FUNCTION_BLOCK MoverList EXTENDS Objective IMPLEMENTS iMoverList
VAR_INPUT
END_VAR
VAR_OUTPUT
END_VAR
VAR
END_VAR

METHOD ActivateAllTrack : BOOL
VAR_INPUT
	Track	: REFERENCE TO Track;
END_VAR
VAR
    i : ULINT;
END_VAR
// this method is not chainable
// monitor .IsAllTrackReady before calling additional commands on this list

// For every valid mover in the list, pass it a ActivateTrack command
FOR i := 1 TO SIZEOF(internalRegisteredMovers) / SIZEOF(internalRegisteredMovers[1]) DO

    IF internalRegisteredMovers[i] <> 0 THEN
        internalRegisteredMovers[i]^.ActivateTrack(Track);
    END_IF

END_FOR
END_METHOD

PROPERTY AllMovers : ARRAY[1..Param.MAX_MOVERS] OF POINTER TO Mover
GET
VAR
	i: ULINT;
	destIndex : ulint;
END_VAR
// returns a front-end-loaded array of pointers to movers in the current mover list
// set up the destination index
destIndex := 1;

// test all the movers
FOR i := 1 TO Param.MAX_MOVERS DO
	// if there's a mover add it to the return value
	IF (internalRegisteredMovers[i] <> 0) THEN
		AllMovers[destIndex] := internalRegisteredMovers[i];
		// increment the destination index
		destIndex := destIndex + 1;
	END_IF;
END_FOR
END_GET
END_PROPERTY

METHOD ApplyAllParameterSet : iMoverList
VAR_INPUT
	ParameterSet		: MotionParameters_typ;
END_VAR

VAR
	i: ULINT;
END_VAR

FOR i := 1 TO SIZEOF( internalRegisteredMovers ) / SIZEOF( internalRegisteredMovers[1] ) DO
	
	IF internalRegisteredMovers[i] <> 0 THEN
		internalRegisteredMovers[i]^.MotionParameters		:= ParameterSet;
	END_IF
	
END_FOR

ApplyAllParameterSet		:= THIS^;
END_METHOD

METHOD Contains : BOOL
VAR_INPUT
	
	Mover		: REFERENCE TO Mover;

END_VAR

VAR
	i: UDINT;
END_VAR


// Check if the input Mover is contained within the existing list
FOR i := 1 TO SIZEOF( internalRegisteredMovers ) / SIZEOF( internalRegisteredMovers[1]) DO
	IF internalRegisteredMovers[i] <> 0 AND internalRegisteredMovers[i] = ADR( Mover ) THEN
		Contains	:= TRUE;
	END_IF
END_FOR
END_METHOD

METHOD DisableAll : iMoverList
VAR
	i		: ULINT;
END_VAR


// For every valid mover in the list, Enable it

FOR i := 1 TO SIZEOF( internalRegisteredMovers ) / SIZEOF( internalRegisteredMovers[1] ) DO
	
	IF internalRegisteredMovers[i] <> 0 THEN
		internalRegisteredMovers[i]^.Disable();
	END_IF

END_FOR

DisableAll	:= THIS^;
END_METHOD

METHOD EnableAll : iMoverList
VAR
	i		: ULINT;
END_VAR


// For every valid mover in the list, Enable it

FOR i := 1 TO SIZEOF( internalRegisteredMovers ) / SIZEOF( internalRegisteredMovers[1] ) DO
	
	IF internalRegisteredMovers[i] <> 0 THEN
		internalRegisteredMovers[i]^.Enable();
	END_IF

END_FOR

EnableAll	:= THIS^;
END_METHOD

METHOD FilterDestinationStation : iMoverList
VAR_INPUT
	Destination	: REFERENCE TO Station;
END_VAR
VAR
	i : ulint;
END_VAR
// filters this mover list for movers that have the stated destination station
FOR i := 1 TO SIZEOF(internalRegisteredMovers) / SIZEOF(internalRegisteredMovers[1]) DO

	// test for valid mover
    IF internalRegisteredMovers[i] <> 0 THEN
		// test for track ready
		IF internalRegisteredMovers[i]^.IsTrackReady THEN
			// unregister this mover if the track id, movetype or destination position do not match
			IF internalRegisteredMovers[i]^.CurrentDestinationTrack <> Destination.TrackId OR
			 internalRegisteredMovers[i]^.CurrentMoveType <> MOVETYPE_STATION OR
			 internalRegisteredMovers[i]^.CurrentDestinationPosition <> Destination.Position THEN
				// unregister this mover, the manual way
				internalRegisteredMovers[i]  := 0; // remove the pointer
                internalRegisteredMoverCount := internalRegisteredMoverCount - 1;
			 END_IF;
		ELSE
			// track was not ready, unregister this mover
			// the manual way
			internalRegisteredMovers[i]  := 0; // remove the pointer
			internalRegisteredMoverCount := internalRegisteredMoverCount - 1;
		END_IF;
	END_IF
	
END_FOR;

// return this list for chaining
FilterDestinationStation := THIS^;
END_METHOD

METHOD GetMoverByLocation : REFERENCE TO Mover
VAR_INPUT
	Index			: USINT;				// 1 is find the first closest mover, 2 is find the second closest mover, 3 is find the third, etc. etc. etc.
	Position		: LREAL;				// fixed track position from which to search for movers by proximity
	Direction		: Tc2_MC2.MC_Direction;	// Positive = find the most positive mover whose position is less than the Input. Negative = find the most negative mover whose position is greater than the Input.		
END_VAR

VAR
	sortState			: USINT;

	StartBuffer			: ARRAY[1..Param.MAX_MOVERS] OF POINTER TO Mover;	// Initial unsorted array of movers
	HoldingBuffer		: ARRAY[1..Param.MAX_MOVERS] OF POINTER TO Mover;	// Holding buffer for sorting operations
	SortBuffer			: ARRAY[1..Param.MAX_MOVERS] OF POINTER TO Mover;	// Fully sorted output buffer
	
	n					: UDINT;	// index var for loops
	location			: UDINT := 1;	// index for placing in Start Buffer without gaps
	moverCount			: UDINT;	// number of movers present in the array
	
	place				: UDINT	:= 1;	// placement index
	level				: UDINT := 1;	// level tracker
	element				: UDINT := 1;	// index tracker
	
	allsorted			: BOOL;		// status bit, array has been successfully sorted
	elementsorted		: BOOL;		// status bit, element has been successfully sorted
	
	nom_size			: UDINT;	// nominal size of elements at this level
	act_size			: UDINT;		// actual size of this sortation element. possibly smaller at the end of the array
	low					: UDINT;	// starting point for index i within this element
	middle				: UDINT;	// starting point for index j within this element
	high				: UDINT;	// end of the sortation merge element at this level, element
	
	i					: UDINT;		// index variable within the merge element
	j					: UDINT;		// index variable within the merge element	
	
	directionalDistance_i		: LREAL;
	directionalDistance_j		: LREAL;
	
	cycles				: UDINT;

END_VAR
// Method is implemented using a Mergesort, for improved performance on systems with high mover counts.

// memcpy( ADR( StartBuffer ), ADR( internalRegisteredMovers ), SIZEOF( internalRegisteredMovers ));

WHILE allsorted = FALSE DO
	
	cycles	:= cycles + 1;
	
	CASE sortState OF
		0:	// ---------------------- Count the number of registered movers & populate StartBuffer without gaps
		
			FOR n := 1 TO ( SIZEOF( internalRegisteredMovers ) / SIZEOF( internalRegisteredMovers[1] ) ) DO
				IF internalRegisteredMovers[n] <> 0 THEN
					moverCount		:= moverCount + 1;
					memcpy( ADR( StartBuffer[location] ), ADR( internalRegisteredMovers[n] ), SIZEOF( internalRegisteredMovers[n] ));
					location		:= location + 1;
				END_IF
			END_FOR
			
			memcpy( ADR( SortBuffer ), ADR( StartBuffer ), SIZEOF( StartBuffer ));
			
			sortState		:= 1;		
		
		1:	// ---------------------- Calculate sortation parameters for the current merge element
		
			nom_size			:= LREAL_TO_UDINT(EXPT( 2, level ));
			
			low					:= ( element - 1 ) * nom_size + 1;
			middle				:= MIN(( low + LREAL_TO_UDINT( FLOOR( nom_size / 2 ))), moverCount );
			high				:= MIN(( low + nom_size - 1), moverCount );
			
			act_size			:= high - low + 1;
			
			i					:= low;
			j					:= middle;
			
			sortState			:= 2;
			
		2:	// ---------------------- Check if the level is completely sorted/merged 
		
			// if nom_size from last level was larger than the number of movers, we are fully sorted
			IF element = 1 AND LREAL_TO_UDINT(EXPT(2,level-1)) > moverCount THEN
				allsorted		:= TRUE;
			// if low is greater than moverCount, we've completed a merge level. increment
			ELSIF low >  moverCount THEN
				memset( ADR( HoldingBuffer ), 0, SIZEOF( HoldingBuffer ));
				level			:= level + 1;
				element			:= 1;
				place			:= 1;
				sortState		:= 1;			
			// i and j are both sortable- move on to direct comparisons			
			ELSE
				sortState		:= 3;	
			END_IF			
			
		3:	// ---------------------- Check if the elements at the indices are sortable or if we're beyond the array
		
			IF ( i >= middle OR i > moverCount ) AND ( j > high OR j > moverCount ) THEN
				// i and j have both reached the end of the merge element
				memcpy( ADR( SortBuffer[low] ), ADR( HoldingBuffer[low] ), act_size * SIZEOF( HoldingBuffer[1] )); 
				element			:= element + 1;
				sortState		:= 1;
			ELSE
				sortState		:= 4;
			END_IF
			
		4:	// ---------------------- Merge elements at indices i & j

			// Calculate directional distances at i & j
			IF Direction = MC_Positive_Direction THEN
				// Calculate for i
				IF ( SortBuffer[i] <> 0 AND i <= moverCount ) AND_THEN SortBuffer[i]^.TrackInfo.TrackPosition <= Position THEN
					directionalDistance_i		:= Position - SortBuffer[i]^.TrackInfo.TrackPosition;
				ELSIF ( SortBuffer[i] <> 0 AND i <= moverCount ) AND_THEN SortBuffer[i]^.TrackInfo.TrackPosition > Position THEN
					directionalDistance_i		:= Position + ( SortBuffer[i]^.CurrentTrack^.Length - SortBuffer[i]^.TrackInfo.TrackPosition );
				END_IF;	
				// Calculate for j
				IF ( SortBuffer[j] <> 0 AND j <= moverCount ) AND_THEN SortBuffer[j]^.TrackInfo.TrackPosition <= Position THEN
					directionalDistance_j		:= Position - SortBuffer[j]^.TrackInfo.TrackPosition;
				ELSIF ( SortBuffer[j] <> 0 AND j <= moverCount ) AND_THEN SortBuffer[j]^.TrackInfo.TrackPosition > Position THEN
					directionalDistance_j		:= Position + ( SortBuffer[j]^.CurrentTrack^.Length - SortBuffer[j]^.TrackInfo.TrackPosition );					 
				END_IF
				
			ELSIF Direction = MC_Negative_Direction THEN
				
				// Calculate for i
				IF  ( SortBuffer[i] <> 0 AND i <= moverCount ) AND_THEN SortBuffer[i]^.TrackInfo.TrackPosition <= Position THEN
					directionalDistance_i		:= SortBuffer[i]^.TrackInfo.TrackPosition + ( SortBuffer[i]^.CurrentTrack^.Length - Position );
				ELSIF  ( SortBuffer[i] <> 0 AND i <= moverCount ) AND_THEN SortBuffer[i]^.TrackInfo.TrackPosition > Position THEN
					directionalDistance_i		:= SortBuffer[i]^.TrackInfo.TrackPosition - Position;
				END_IF
				// Calculate for j
				IF ( SortBuffer[j] <> 0 AND j <= moverCount ) AND_THEN SortBuffer[j]^.TrackInfo.TrackPosition <= Position THEN
					directionalDistance_j		:= SortBuffer[j]^.TrackInfo.TrackPosition + ( SortBuffer[j]^.CurrentTrack^.Length - Position );
				ELSIF ( SortBuffer[j] <> 0 AND j <= moverCount ) AND_THEN SortBuffer[j]^.TrackInfo.TrackPosition > Position THEN
					directionalDistance_j		:= SortBuffer[j]^.TrackInfo.TrackPosition - Position;
				END_IF
				
			ELSE
				// closest in any direction, typically for linear, non-modulo tracks
				IF ( SortBuffer[i] <> 0 AND i <= moverCount ) THEN
					directionalDistance_i		:= ABS(SortBuffer[i]^.TrackInfo.TrackPosition - Position);
				END_IF
				IF ( SortBuffer[j] <> 0 AND j <= moverCount ) THEN
					directionalDistance_j		:= ABS(SortBuffer[j]^.TrackInfo.TrackPosition - Position);
				END_IF
				
			END_IF
			
			// If j alone is beyond a sortable range, grab i
			IF j > high OR j > moverCount THEN
				HoldingBuffer[place]		:= SortBuffer[i];
				place						:= place + 1;
				i							:= i + 1;
			// If i is beyond a sortable range, grab j
			ELSIF i >= middle OR i > moverCount THEN
				HoldingBuffer[place]		:= SortBuffer[j];
				place						:= place + 1;
				j							:= j + 1;
			ELSIF directionalDistance_i <= directionalDistance_j THEN
				HoldingBuffer[place]		:= SortBuffer[i];
				place						:= place + 1;
				i							:= i + 1;
			ELSIF directionalDistance_j < directionalDistance_i THEN
				HoldingBuffer[place]		:= SortBuffer[j];
				place						:= place + 1;
				j							:= j + 1;					
			END_IF
			
			sortState		:= 3;
			
	END_CASE
END_WHILE

IF Index < 1 OR Index > THIS^.RegisteredMoverCount THEN
	GetMoverByLocation REF= 0;
ELSE
	GetMoverByLocation REF= SortBuffer[Index]^;
END_IF

IF __ISVALIDREF(GetMoverByLocation) = FALSE THEN
	ErrorMover.SourceInstancePath		:= THIS^.InstancePath;
	GetMoverByLocation					REF= ErrorMover;
END_IF
END_METHOD

METHOD HaltAll : iMoverList
VAR
	i		: ULINT;
END_VAR


// For every valid mover in the list, Halt it

FOR i := 1 TO SIZEOF( internalRegisteredMovers ) / SIZEOF( internalRegisteredMovers[1] ) DO
	
	IF internalRegisteredMovers[i] <> 0 THEN
		internalRegisteredMovers[i]^.Halt();
	END_IF

END_FOR

HaltAll	:= THIS^;
END_METHOD

PROPERTY IsAllMoversDisabled : bool
GET
VAR
	i: ULINT;
END_VAR
IsAllMoversDisabled		:= TRUE;		// ...default

FOR i := 1 TO SIZEOF( internalRegisteredMovers ) / SIZEOF( internalRegisteredMovers[1] ) DO

	IF internalRegisteredMovers[i] <> 0 AND_THEN internalRegisteredMovers[i]^.Ready = TRUE THEN
		IsAllMoversDisabled		:= FALSE;
	END_IF;


END_FOR
END_GET
END_PROPERTY

PROPERTY IsAllMoversHalted : BOOL
GET
VAR
	i: ULINT;
END_VAR
IsAllMoversHalted		:= TRUE;		// ...default

FOR i := 1 TO SIZEOF( internalRegisteredMovers ) / SIZEOF( internalRegisteredMovers[1] ) DO
	// check for valid mover
	IF internalRegisteredMovers[i] <> 0 AND_THEN internalRegisteredMovers[i]^.AxisReference.Status.Moving = TRUE THEN
		IsAllMoversHalted		:= FALSE;
	END_IF;

END_FOR
END_GET
END_PROPERTY

PROPERTY IsAllMoversReady : BOOL
GET
VAR
	i: ULINT;
END_VAR

IsAllMoversReady		:= TRUE;		// ...default

FOR i := 1 TO SIZEOF( internalRegisteredMovers ) / SIZEOF( internalRegisteredMovers[1] ) DO

	IF internalRegisteredMovers[i] <> 0 AND_THEN internalRegisteredMovers[i]^.Ready = FALSE THEN
		IsAllMoversReady		:= FALSE;
	END_IF;

END_FOR
END_GET
END_PROPERTY

PROPERTY IsAllTrackReady : BOOL
GET
VAR
	i : ULINT;
	size : ULINT;
	allReady : BOOL;
	zeroCount : ULINT;
END_VAR
// For every valid mover in the list, sum up IsTrackReady
// intentionally returns false if no movers are found
// this is to support the typical use case when MoverList.ActivateAllTrack and .IsAllTrackReady are called back-to-back
// to peroform a track change
// this ensures that during the ~20ms track change in software when no movers may be present on the track, this response will not inadvertantly advance code
// if zero movers is a common situation an OR condition of "MoverList.RegisteredMoverCount = 0" can be added to the statement calling this
allReady := TRUE;
size := SIZEOF(internalRegisteredMovers) / SIZEOF(internalRegisteredMovers[1]);
zeroCount := 0;

FOR i := 1 TO size DO

    IF internalRegisteredMovers[i] <> 0 THEN
        allReady := allReady AND internalRegisteredMovers[i]^.IsTrackReady;
	ELSE
		zeroCount := zeroCount + 1;
    END_IF

END_FOR

// check for no movers
IF zeroCount = (size) THEN
	allReady := FALSE;
END_IF

IsAllTrackReady := allReady; // return result
END_GET
END_PROPERTY

PROPERTY IsNoMoverBusy : BOOL
GET
VAR
		i: ULINT;
END_VAR
IsNoMoverBusy		:= TRUE;		// ...default

FOR i := 1 TO SIZEOF( internalRegisteredMovers ) / SIZEOF( internalRegisteredMovers[1] ) DO
	// check for valid mover
	IF internalRegisteredMovers[i] <> 0 AND_THEN internalRegisteredMovers[i]^.Busy = TRUE THEN
		IsNoMoverBusy		:= FALSE;
	END_IF;

END_FOR
END_GET
END_PROPERTY

METHOD LogicalComplement : MoverList
VAR_INPUT
END_VAR

VAR
	i: UINT;
END_VAR


FOR i := 1 TO Param.MAX_MOVERS DO
	
	IF NOT THIS^.Contains( Mediator.MoverArray[i]^ ) THEN
		LogicalComplement.RegisterMover( Mediator.MoverArray[i]^ );
	END_IF

END_FOR
END_METHOD

METHOD LogicalDifference : MoverList
VAR_INPUT
	
	MoverList		: MoverList;

END_VAR
VAR
	i				: UINT;
END_VAR



FOR i := 1 TO Param.MAX_MOVERS DO
	
	IF THIS^.Contains( Mediator.MoverArray[i]^ ) AND NOT MoverList.Contains( Mediator.MoverArray[i]^ ) THEN
		LogicalDifference.RegisterMover( Mediator.MoverArray[i]^ );
	END_IF

END_FOR
END_METHOD

METHOD LogicalIntersect : MoverList
VAR_INPUT
	
	MoverList		: MoverList;

END_VAR

VAR
	i				: UINT;
END_VAR


FOR i := 1 TO Param.MAX_MOVERS DO
	
	IF MoverList.Contains( Mediator.MoverArray[i]^ ) AND THIS^.Contains( Mediator.MoverArray[i]^ ) THEN
		LogicalIntersect.RegisterMover( Mediator.MoverArray[i]^ );	
	END_IF
	
END_FOR
END_METHOD

METHOD LogicalUnion : MoverList
VAR_INPUT
	
	MoverList		: MoverList;

END_VAR


LogicalUnion.RegisterMoverList( MoverList );
LogicalUnion.RegisterMoverList( THIS^ );
END_METHOD

METHOD MoveAllToPosition : iMoverList
VAR_INPUT

    DestinationPosition : LREAL; // position on track for all shuttles to move towards	

END_VAR

VAR
    i : ulint;
END_VAR
// For every valid mover in the list, pass it a MoveToPosition command
FOR i := 1 TO SIZEOF(internalRegisteredMovers) / SIZEOF(internalRegisteredMovers[1]) DO

    IF internalRegisteredMovers[i] <> 0 THEN
        internalRegisteredMovers[i]^.MoveToPosition(DestinationPosition);
    END_IF

END_FOR

MoveAllToPosition := THIS^; // return this, to allow method chaining
END_METHOD

METHOD MoveAllToStation : iMoverList
VAR_INPUT

    DestinationStation : REFERENCE TO Station;

END_VAR

VAR
    i : ULINT;
END_VAR
// For every valid mover in the list, pass it a MoveToStation command
FOR i := 1 TO SIZEOF(internalRegisteredMovers) / SIZEOF(internalRegisteredMovers[1]) DO

    IF internalRegisteredMovers[i] <> 0 THEN
        internalRegisteredMovers[i]^.MoveToStation(DestinationStation);
    END_IF

END_FOR

MoveAllToStation := THIS^; // allows method chaining
END_METHOD

METHOD MoveAllVelocity : iMoverList
VAR_INPUT

    Velocity : LREAL;

END_VAR
VAR
    i : ULINT;
END_VAR
// For every valid mover in the list, pass it a MoveVelocity command
FOR i := 1 TO SIZEOF(internalRegisteredMovers) / SIZEOF(internalRegisteredMovers[1]) DO

    IF internalRegisteredMovers[i] <> 0 THEN
        internalRegisteredMovers[i]^.MoveVelocity(Velocity);
    END_IF

END_FOR

MoveAllVelocity := THIS^;
END_METHOD

METHOD SetAllAcceleration : iMoverList
VAR_INPUT

    Acceleration : LREAL;

END_VAR

VAR
    i : ULINT;
END_VAR
// For every valid mover in the list, set the Acceleration values
FOR i := 1 TO SIZEOF(internalRegisteredMovers) / SIZEOF(internalRegisteredMovers[1]) DO

    IF internalRegisteredMovers[i] <> 0 THEN
        internalRegisteredMovers[i]^.SetAcceleration(Acceleration);
    END_IF

END_FOR

SetAllAcceleration := THIS^;
END_METHOD

METHOD SetAllDeceleration : iMoverList
VAR_INPUT

    Deceleration : LREAL;

END_VAR
VAR
    i : ULINT;
END_VAR
// For every valid mover in the list, set the Deceleration values
FOR i := 1 TO SIZEOF(internalRegisteredMovers) / SIZEOF(internalRegisteredMovers[1]) DO

    IF internalRegisteredMovers[i] <> 0 THEN
        internalRegisteredMovers[i]^.SetDeceleration(Deceleration);
    END_IF

END_FOR

SetAllDeceleration := THIS^;
END_METHOD

METHOD SetAllDirection : iMoverList
VAR_INPUT

    Direction : Tc3_Mc3Definitions.MC_DIRECTION;

END_VAR
VAR
    i : ULINT;
END_VAR
// For every valid mover in the list, update the internal Direction parameter
FOR i := 1 TO SIZEOF(internalRegisteredMovers) / SIZEOF(internalRegisteredMovers[1]) DO

    IF internalRegisteredMovers[i] <> 0 THEN
        internalRegisteredMovers[i]^.SetDirection(Direction);
    END_IF

END_FOR

SetAllDirection := THIS^;
END_METHOD

METHOD SetAllGap : iMoverList
VAR_INPUT
    Gap : LREAL;
END_VAR
VAR
    i : ULINT;
END_VAR
// For every valid mover in the list, update the internal Gap Parameter
FOR i := 1 TO SIZEOF(internalRegisteredMovers) / SIZEOF(internalRegisteredMovers[1]) DO

    IF internalRegisteredMovers[i] <> 0 THEN
        internalRegisteredMovers[i]^.SetGap(Gap);
    END_IF

END_FOR

SetAllGap := THIS^;
END_METHOD

METHOD SetAllGapMode : iMoverList
VAR_INPUT
    Mode	: MC_GAP_CONTROL_MODE;
END_VAR
VAR
    i : ULINT;
END_VAR
// For every valid mover in the list, update the internal GapMode Parameter
FOR i := 1 TO SIZEOF(internalRegisteredMovers) / SIZEOF(internalRegisteredMovers[1]) DO

    IF internalRegisteredMovers[i] <> 0 THEN
        internalRegisteredMovers[i]^.SetGapMode(Mode);
    END_IF

END_FOR

SetAllGapMode := THIS^;
END_METHOD

METHOD SetAllJerk : iMoverList
VAR_INPUT

    Jerk : LREAL;

END_VAR
VAR
    i : ULINT;
END_VAR
// For every valid mover in the list, update the internal Jerk Parameter
FOR i := 1 TO SIZEOF(internalRegisteredMovers) / SIZEOF(internalRegisteredMovers[1]) DO

    IF internalRegisteredMovers[i] <> 0 THEN
        internalRegisteredMovers[i]^.SetJerk(Jerk);
    END_IF

END_FOR

SetAllJerk := THIS^;
END_METHOD

METHOD SetAllVelocity : iMoverList
VAR_INPUT

    Velocity : LREAL;

END_VAR
VAR
    i : ULINT;
END_VAR
// For every valid mover in the list, set the Velocity values
FOR i := 1 TO SIZEOF(internalRegisteredMovers) / SIZEOF(internalRegisteredMovers[1]) DO

    IF internalRegisteredMovers[i] <> 0 THEN
        internalRegisteredMovers[i]^.SetVelocity(Velocity);
    END_IF

END_FOR

SetAllVelocity := THIS^;
END_METHOD

END_FUNCTION_BLOCK

(* stored: Version 1.1.0.1, ProductVersion 3.1.4026.12
   POU MoverList: Id {6a6492c3-5dac-4c49-8708-8eab34cf4a1d}, SpecialFunc None
   Folder Methods: Id {f0610894-1931-4d0e-a817-1d1b4c8212b1}
   Folder Properties: Id {3fdda14a-1516-48f6-a734-917962304085}
   Method ActivateAllTrack: Id {ad8953ff-aa85-09f3-0f73-09c72fab1fb2}
   Property AllMovers: Id {52a1695b-1d8f-0ef9-3cd3-1395c39cd0c3}
   Get Get: Id {ef34fbdc-dfde-05ba-0251-c668ef47ba93}
   Method ApplyAllParameterSet: Id {ee27996d-bc19-0617-3aa0-2b2a5832f4d1}
   Method Contains: Id {49bffcb6-3630-0c15-279c-3e0d2426245a}
   Method DisableAll: Id {34930db0-7d57-0ea7-09de-0bf399bd6e52}
   Method EnableAll: Id {99b09009-74d0-0637-0d16-bcb874d15a8e}
   Method FilterDestinationStation: Id {c0547a1c-2297-0060-3112-c0f3bffc12c0}
   Method GetMoverByLocation: Id {2ed381fa-32e4-0a91-0551-8d2b2515ae32}
   Method HaltAll: Id {da08056b-7ab2-0f88-0878-dde248efd6e3}
   Property IsAllMoversDisabled: Id {62b7d526-7474-0452-005a-29acf2e3f507}
   Get Get: Id {65b9f9db-b175-0367-29fb-c0545e966bd7}
   Property IsAllMoversHalted: Id {7eaef20f-f1ea-0872-0da2-c36e439864d5}
   Get Get: Id {d65b9e73-d62f-07d0-2566-ad06acb540ed}
   Property IsAllMoversReady: Id {60630f08-9378-0450-0bc7-1b90b2e15524}
   Get Get: Id {bc6cb727-5d1a-0db0-2b04-cbe3e5287984}
   Property IsAllTrackReady: Id {6e2cc0c2-f637-0149-0661-22b5c671a702}
   Get Get: Id {cf4fcf50-2d73-046b-2dbd-7c13f3f0f631}
   Property IsNoMoverBusy: Id {cece049b-4403-0dbb-1591-1117ce3abf4b}
   Get Get: Id {31873de7-e1fb-04a5-1fa5-4b95bfc590a7}
   Method LogicalComplement: Id {d6bb64e7-1c08-0ac2-2a32-42be336ae034}
   Method LogicalDifference: Id {a0c51d7c-09ca-0254-378e-53c1775ec0b5}
   Method LogicalIntersect: Id {83ddeada-4967-0249-0f08-a02d5e1843f1}
   Method LogicalUnion: Id {328a0d90-4052-09a0-1fd6-2c3bd426e573}
   Method MoveAllToPosition: Id {bd912cae-8475-45f4-9366-6d4e3f45dbfd}
   Method MoveAllToStation: Id {7e8649c5-afae-438c-9d7c-0849d9778d85}
   Method MoveAllVelocity: Id {374fc66e-e454-42d2-84eb-da107ea5cc5b}
   Method SetAllAcceleration: Id {e13ce26b-c052-44c4-b781-edc2323e6bd8}
   Method SetAllDeceleration: Id {b4a74589-da0f-40fe-9d74-9df176d68d9e}
   Method SetAllDirection: Id {61dc841d-816d-4126-817b-0edc70c354b4}
   Method SetAllGap: Id {1311da71-cec2-0375-2ed8-ab2381f7cc99}
   Method SetAllGapMode: Id {eb4b4f5b-2a13-0c63-3742-71822424864a}
   Method SetAllJerk: Id {713a2faa-4d72-4826-b835-2931c44827b9}
   Method SetAllVelocity: Id {cee9569c-3982-4955-90f1-8e5baf09c135} *)
